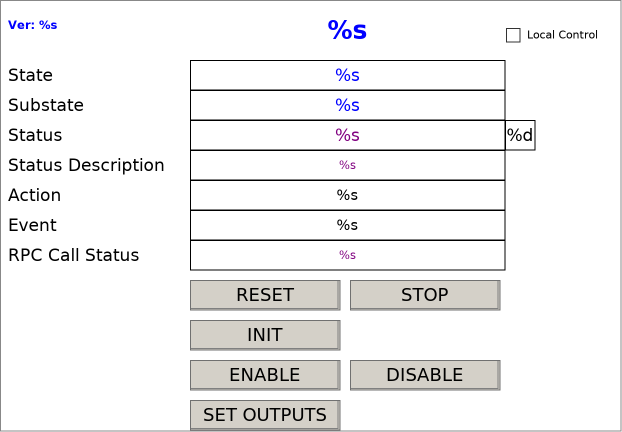
VISUALIZATION GUI_TEMPLATE_IODEV  // 622x432
VAR_IN_OUT
	m_Instance:	FB_IODEV_BASE;
END_VAR
    Rectangle (190,60 315x30), "%s", text variable: m_Instance.stat.sState
    Rectangle (190,90 315x30), "%s", text variable: m_Instance.stat.sSubstate
    Button (190,280 150x30), "RESET", input disabled if: (m_Instance.stat.bLocal = FALSE) <> 0
        OnMouseDown: execute { m_Instance.ctrl.nCommand := E_IODEV_COMMAND.RESET; m_Instance.ctrl.bExecute := TRUE; }
    Button (190,320 150x30), "INIT", input disabled if: (m_Instance.stat.bLocal = FALSE) <> 0
        OnMouseDown: execute { m_Instance.ctrl.nCommand := E_IODEV_COMMAND.INIT; m_Instance.ctrl.bExecute := TRUE; }
    Button (350,280 150x30), "STOP", input disabled if: (m_Instance.stat.bLocal = FALSE) <> 0
        OnMouseDown: execute { m_Instance.ctrl.nCommand := E_IODEV_COMMAND.STOP; m_Instance.ctrl.bExecute := TRUE; }
    Button (190,360 150x30), "ENABLE", input disabled if: (m_Instance.stat.bLocal = FALSE) <> 0
        OnMouseDown: execute { m_Instance.ctrl.nCommand := E_IODEV_COMMAND.ENABLE; m_Instance.ctrl.bExecute := TRUE; }
    Button (350,360 150x30), "DISABLE", input disabled if: (m_Instance.stat.bLocal = FALSE) <> 0
        OnMouseDown: execute { m_Instance.ctrl.nCommand := E_IODEV_COMMAND.DISABLE; m_Instance.ctrl.bExecute := TRUE; }
    Button (190,400 150x30), "SET OUTPUTS", input disabled if: (m_Instance.stat.bLocal = FALSE) <> 0
        OnMouseClick: execute { m_Instance.ctrl.nCommand := E_IODEV_COMMAND.SET_OUTPUTS; m_Instance.ctrl.bExecute := TRUE; }
    Rectangle (5,60 180x30), "State"
    Rectangle (5,90 180x30), "Substate"
    Rectangle (190,120 315x30), "%s", text variable: m_Instance.stat.sStatus
    Rectangle (190,150 315x30), "%s", text variable: m_Instance.stat.sErrorText
    Rectangle (5,120 180x30), "Status"
    Rectangle (5,150 180x30), "Status Description"
    Rectangle (190,180 315x30), "%s", text variable: m_Instance.stat.sActionDesc
    Rectangle (190,210 315x30), "%s", text variable: m_Instance.stat.sEventDesc
    Rectangle (5,180 180x30), "Action"
    Rectangle (5,210 180x30), "Event"
    Rectangle (190,12 315x35), "%s", text variable: m_Instance.cfg.sName
    Rectangle (505,120 30x30), "%d", text variable: m_Instance.stat.nStatus
    Checkbox (504,20 116x30), "Local Control", variable: m_Instance.stat.bLocal
    Rectangle (190,240 315x30), "%s", text variable: m_Instance.stat.sRPCErrorText
    Rectangle (5,240 180x30), "RPC Call Status"
    Rectangle (5,10 99x30), "Ver: %s", tooltip "'IODev.library version'", text variable: m_Instance.stat.sLibVersion, input disabled if: true
END_VISUALIZATION

(* stored: Version 1.1.0.1, ProductVersion 3.1.4022.16
   Visu GUI_TEMPLATE_IODEV: Id {208abcb1-f1a3-4a00-92a5-f362cd7556ac} *)
